// TIA Portal V20 export
VAR_GLOBAL   // PLC tag table "Sonplas_Outputs"
   DQ_SonplasDiagDPCoupler AT %Q200.0 : Bool;
   DQ_SonplasReady AT %Q200.1 : Bool;
   DQ_SonplasNoEStop AT %Q200.2 : Bool;
   DQ_SonplasDoorsClosed AT %Q200.3 : Bool;
   DQ_SonplasRunError AT %Q200.4 : Bool;
   DQ_SonplasFreeQ200_5 AT %Q200.5 : Bool;
   DQ_SonplasFreeQ200_6 AT %Q200.6 : Bool;
   DQ_SonplasFreeQ200_7 AT %Q200.7 : Bool;
   DQ_SonplasFreeQ201_0 AT %Q201.0 : Bool;
   DQ_SonplasFreeQ201_1 AT %Q201.1 : Bool;
   DQ_SonplasFreeQ201_2 AT %Q201.2 : Bool;
   DQ_SonplasFreeQ201_3 AT %Q201.3 : Bool;
   DQ_SonplasFreeQ201_4 AT %Q201.4 : Bool;
   DQ_SonplasFreeQ201_5 AT %Q201.5 : Bool;
   DQ_SonplasFreeQ201_6 AT %Q201.6 : Bool;
   DQ_SonplasFreeQ201_7 AT %Q201.7 : Bool;
   DQ_SonplasShuttle1InPos AT %Q202.0 : Bool;
   DQ_SonplasFreeQ202_1 AT %Q202.1 : Bool;
   DQ_SonplasFreeQ202_2 AT %Q202.2 : Bool;
   DQ_SonplasFreeQ202_3 AT %Q202.3 : Bool;
   DQ_SonplasFreeQ202_4 AT %Q202.4 : Bool;
   DQ_SonplasFreeQ202_5 AT %Q202.5 : Bool;
   DQ_SonplasPart1OK AT %Q202.6 : Bool;
   DQ_SonplasPart1NOK AT %Q202.7 : Bool;
   DQ_SonplasShuttle2InPos AT %Q203.0 : Bool;
   DQ_SonplasFreeQ203_1 AT %Q203.1 : Bool;
   DQ_SonplasFreeQ203_2 AT %Q203.2 : Bool;
   DQ_SonplasFreeQ203_3 AT %Q203.3 : Bool;
   DQ_SonplasFreeQ203_4 AT %Q203.4 : Bool;
   DQ_SonplasFreeQ203_5 AT %Q203.5 : Bool;
   DQ_SonplasPart2OK AT %Q203.6 : Bool;
   DQ_SonplasPart2NOK AT %Q203.7 : Bool;
   DQ_SonplasResultAccepted AT %Q244.0 : Bool;
   DQ_SonplasFreeQ244_1 AT %Q244.1 : Bool;
   DQ_SonplasFreeQ244_2 AT %Q244.2 : Bool;
   DQ_SonplasFreeQ244_3 AT %Q244.3 : Bool;
   DQ_SonplasFreeQ244_4 AT %Q244.4 : Bool;
   DQ_SonplasFreeQ244_5 AT %Q244.5 : Bool;
   DQ_SonplasFreeQ244_6 AT %Q244.6 : Bool;
   DQ_SonplasFreeQ244_7 AT %Q244.7 : Bool;
   AQ_SonplasDMC_Code1 AT %QB204 : Byte;
   AQ_SonplasDMC_Code2 AT %QB224 : Byte;
END_VAR
